{attribute 'linkalways'} 
{attribute 'no_explicit_call' := 'This FB is a CLASS and must be accessed using methods or properties'}
{attribute 'enable_dynamic_creation'}
FUNCTION_BLOCK GraphApi IMPLEMENTS I_RpcApi, I_HostGraphs, I_EventEmitter
VAR
	graphFramework : I_GraphFramework;
	eventEmitter : EventEmitter;
	graphHost : GraphHost(THIS^, eventEmitter);
	loadGraphRpcHandler : LoadGraphRpcHandler;
	multiUserLoadGraphRpcHandler : MultiUserLoadGraphRpcHandler;
	getBlueprintsRpcHandler : GetBlueprintsRpcHandler;
	getDatatypesRpcHandler : GetDatatypesRpcHandler;
	getContentValueHandler : GetContentValueHandler;
END_VAR

METHOD FB_exit : BOOL
VAR_INPUT
	bInCopyCode : BOOL; // if TRUE, the exit method is called for exiting an instance that is copied afterwards (online change).
END_VAR
IF bInCopyCode THEN
	RETURN;
END_IF

graphs.DisposeAll();
END_METHOD

METHOD FB_init : BOOL
VAR_INPUT
	bInitRetains : BOOL; // if TRUE, the retain variables are initialized (warm start / cold start)
	bInCopyCode : BOOL;  // if TRUE, the instance afterwards gets moved into the copy code (online change)
	GraphFramework : I_GraphFramework;
END_VAR
THIS^.graphFramework := GraphFramework;

getBlueprintsRpcHandler.Initialize(GraphFramework.NodeFactory);
getDatatypesRpcHandler.Initialize(GraphFramework.Datatypes);
loadGraphRpcHandler.Initialize(GraphFramework, graphHost);
multiUserLoadGraphRpcHandler.Initialize(GraphFramework, graphHost);
getContentValueHandler.Initialize(graphHost);
END_METHOD

PROPERTY PUBLIC Graphs : I_Graphs
GET
Graphs := graphHost;
END_GET
END_PROPERTY

METHOD PUBLIC OffEvent
VAR_INPUT
	EventName : T_MaxString;
	EventHandler : I_EventHandler;
END_VAR
eventEmitter.OffEvent(EventName, EventHandler);
END_METHOD

METHOD PUBLIC OnceEvent
VAR_INPUT
	EventName : T_MaxString;
	EventHandler : I_EventHandler;
END_VAR
eventEmitter.OnceEvent(EventName, EventHandler);
END_METHOD

METHOD PUBLIC OnEvent
VAR_INPUT
	EventName : T_MaxString;
	EventHandler : I_EventHandler;
END_VAR
eventEmitter.OnEvent(EventName, EventHandler);
END_METHOD

METHOD RegisterWith
VAR_INPUT
	Server : I_RpcServer;
END_VAR
Server.RegisterRpcHandler('LoadGraph',loadGraphRpcHandler);
Server.RegisterRpcHandler('LoadMultiUserGraph',multiUserLoadGraphRpcHandler);
Server.RegisterRpcHandler('GetBlueprints',getBlueprintsRpcHandler);
Server.RegisterRpcHandler('GetDatatypes',getDatatypesRpcHandler);
Server.RegisterRpcHandler('GetContentValue',getContentValueHandler);
END_METHOD

END_FUNCTION_BLOCK

(* stored: Version 1.1.0.1, ProductVersion 3.1.4024.12
   POU GraphApi: Id {2c0ea926-bac0-4e3d-aff9-a56ab39ef9c2}, SpecialFunc None
   Folder Constructor: Id {a5a3a9e0-4cb7-4fba-88b9-60a3e6636f4c}
   Folder Distructor: Id {0fdb84a8-ace4-4238-b174-550597ff2aba}
   Method FB_exit: Id {d9538b94-d79a-4082-86d0-2c014ba7836c}
   Method FB_init: Id {2373ca6b-d93b-4acb-a3d9-5123e1018cb3}
   Property Graphs: Id {e3bdacdc-062d-4bf1-8651-c00274d46505}
   Get Get: Id {5ddb39ce-fbd3-42a2-96b5-4bb5a40d2db3}
   Method OffEvent: Id {d2da028d-1e84-4815-bcc4-d479629ffab3}
   Method OnceEvent: Id {f4b849ab-4690-4f1c-bf7e-033bc47bfc9b}
   Method OnEvent: Id {13ad5aa7-a62d-48a5-be3a-92d4ee18a5ad}
   Method RegisterWith: Id {8110307c-5ce7-4eb2-aa8c-6ce5497795c1} *)
